Yaskawa INFORM job: SHIP-R1.JBI

/JOB
//NAME SHIP-R1
//POS
///NPOS 1,0,0,0,0,0
///TOOL 0
///POSTYPE PULSE
///PULSE
C00000=-2,-200176,-136830,6,-29582,1
//INST
///DATE 2023/08/08 10:16
///ATTR SC,RW
///GROUP1 RB1
NOP
MOVJ C00000 VJ=0.78
END
